{attribute 'linkalways'} 
{attribute 'no_explicit_call' := 'This FB is a CLASS and must be accessed using methods or properties'}
{attribute 'enable_dynamic_creation'}
FUNCTION_BLOCK _DWORD EXTENDS NumericDatatypeBase
VAR
	localData : DWORD;
	activeData : REFERENCE TO DWORD REF= localData;
END_VAR

PROPERTY PUBLIC Address : PVOID
GET
Address := ADR(activeData);
END_GET
END_PROPERTY

METHOD PUBLIC ClearReference
VAR_INPUT
END_VAR
activeData REF= localData;
END_METHOD

METHOD PUBLIC Clone : I_Datatype
VAR
    pClone : POINTER TO _DWORD;
END_VAR
pClone := __NEW(_DWORD(InitialValue := Value));
Clone := pClone^;
END_METHOD

METHOD FB_init : BOOL
VAR_INPUT
	bInitRetains : BOOL; // if TRUE, the retain variables are initialized (warm start / cold start)
	bInCopyCode : BOOL;  // if TRUE, the instance afterwards gets moved WORDo the copy code (online change)
	InitialValue : DWORD;
END_VAR
localData := InitialValue;
END_METHOD

PROPERTY PUBLIC IsFloat : BOOL
GET
IsFloat := FALSE;
END_GET
END_PROPERTY

PROPERTY PUBLIC IsSigned : BOOL
GET
IsSigned := FALSE;
END_GET
END_PROPERTY

METHOD PUBLIC MakeReferenceTo
VAR_INPUT
	ReferenceTarget : REFERENCE TO DWORD;
END_VAR
activeData REF= ReferenceTarget;
END_METHOD

PROPERTY PUBLIC MaxValue : DWORD
GET
MaxValue := DatatypeLimits.DWORD_MAX_VALUE;
END_GET
END_PROPERTY

PROPERTY PUBLIC MinValue : DWORD
GET
MinValue := DatatypeLimits.DWORD_MIN_VALUE;
END_GET
END_PROPERTY

METHOD PROTECTED SerializeMaxValue
VAR_INPUT
	Serializer : I_Serializer;
END_VAR
Serializer.AddDword(MaxValue);
END_METHOD

METHOD PROTECTED SerializeMinValue
VAR_INPUT
	Serializer : I_Serializer;
END_VAR
Serializer.AddDword(MinValue);
END_METHOD

METHOD PUBLIC SerializeWith
VAR_INPUT
	Serializer : I_Serializer;
END_VAR
Serializer.AddDword(activeData);
END_METHOD

PROPERTY PUBLIC Size : UDINT
GET
Size := SIZEOF(activeData);
END_GET
END_PROPERTY

METHOD TryDeserializeFrom : BOOL
VAR_INPUT
	Deserializer : I_Deserializer;
	Feedback : I_DeserializerFeedback;
END_VAR
TryDeserializeFrom := Deserializer.TryGetDword(activeData, Feedback);
END_METHOD

METHOD TryMakeReferenceTo : BOOL
VAR_INPUT
	Target : I_Datatype;
END_VAR
VAR
	pTargetData : POINTER TO DWORD;
END_VAR
IF NOT (Target.TypeName = TypeName) THEN
	RETURN;
END_IF

pTargetData := Target.Address;
activeData REF= pTargetData^;
TryMakeReferenceTo := TRUE;
END_METHOD

PROPERTY PUBLIC TypeName : T_MAXSTRING
GET
TypeName := 'DWORD';
END_GET
END_PROPERTY

PROPERTY PUBLIC Value : DWORD
GET
Value := activeData;
END_GET
SET
activeData := Value;
END_SET
END_PROPERTY

END_FUNCTION_BLOCK

(* stored: Version 1.1.0.1, ProductVersion 3.1.4024.12
   POU _DWORD: Id {a69b5e98-b62a-4b60-88b3-7f05ee8870df}, SpecialFunc None
   Folder Constructor: Id {458b09b5-3458-407e-8700-398f9f921ff6}
   Folder Protected: Id {29138281-226c-406c-ae99-6c29f217a370}
   Property Address: Id {73d27cc8-5e99-49c5-aa77-c5675b0f83eb}
   Get Get: Id {48b57b71-2329-45fd-a075-b72cd3a3fdf5}
   Method ClearReference: Id {7cc2095c-320b-4185-b8ec-803ac28a46d5}
   Method Clone: Id {3c57a5c3-a50c-40c4-8785-22697f43c9c8}
   Method FB_init: Id {ba205e89-de43-42ef-a5c9-9a5728f9ff76}
   Property IsFloat: Id {0582ea1b-81cd-4670-ab27-a189c6176fc3}
   Get Get: Id {88babab9-13e5-4a2e-8e13-dfae403cb947}
   Property IsSigned: Id {f9bb808d-5bd6-46c9-9af3-ca63bae850e0}
   Get Get: Id {2c93fb64-b502-4bde-8665-eaeea81e33d9}
   Method MakeReferenceTo: Id {2758a4c8-0d0d-4d27-b0c0-fd2ab76a7da5}
   Property MaxValue: Id {abce0e7e-cc00-4542-aac4-af03fde4b7c2}
   Get Get: Id {2935896a-0be7-4ae3-886e-ddd656762856}
   Property MinValue: Id {e645042e-cb47-44c8-a198-129e8ddffca3}
   Get Get: Id {bfc36f2d-db52-4d00-bbae-e580fa95ec5e}
   Method SerializeMaxValue: Id {dd2d0615-f6fb-4dbf-97dc-2c94c0e5be6b}
   Method SerializeMinValue: Id {8a0d636a-30e0-4cd4-aa49-d380b02c09a6}
   Method SerializeWith: Id {01a64055-5e70-412c-ad58-78577339351c}
   Property Size: Id {21c9beed-dbf5-4a9a-a440-077dedb1ef32}
   Get Get: Id {70e5c1a7-0b4b-40a2-91f0-0a8bd85baaf5}
   Method TryDeserializeFrom: Id {2b51b55f-b4d4-47bd-ac40-5a3a263732ec}
   Method TryMakeReferenceTo: Id {eba0c1e4-329d-4d2d-9a0c-d746ec51ce46}
   Property TypeName: Id {c7a338e8-859e-44ad-9847-288fd60b7375}
   Get Get: Id {d36513bd-354c-439c-8f1a-77550861b42e}
   Property Value: Id {5548dbe8-e731-4bad-a0ad-2df15646b936}
   Get Get: Id {91b021ee-d3df-453c-a8b2-0397216bcdda}
   Set Set: Id {a8b313c0-afde-4267-8fb8-f313ec35e349} *)
